TYPE ST_OpenLoopControl :
STRUCT
	fBoreArea : LREAL := 0.0033183;
	fAnnulusArea : LREAL := 0.0023562;
	fMaxFlowCapacity : LREAL := 30; //[l/min]
END_STRUCT
END_TYPE

(* stored: Version 1.1.0.1, ProductVersion 3.1.4024.10
   DUT ST_OpenLoopControl: Id {d3ff122b-2654-4a8f-b887-57a35b2cf102} *)
